TYPE "Prod_Beam_Ctrl"
VERSION : 0.1
// Block: Prod_Beam_Ctrl
   STRUCT
      Setup_LinePreparation_Exe : Bool;
      STOP_FineTurno : Bool;
      STOP_ControlloQualita : Bool;
      STOP_End_Of_Production : Bool;
      Beams_Data : Prod_Beam_Data;
   END_STRUCT;

END_TYPE
